// LS Electric XG5000 project: 동남140
// PLC NewPLC
// module base 0 slot 0: 입출력 모듈:XBC-DN/DP14E (DC 24V 입력 8점, 트랜지스터 출력 6점)

PROGRAM NewProgram (task: 스캔 프로그램)

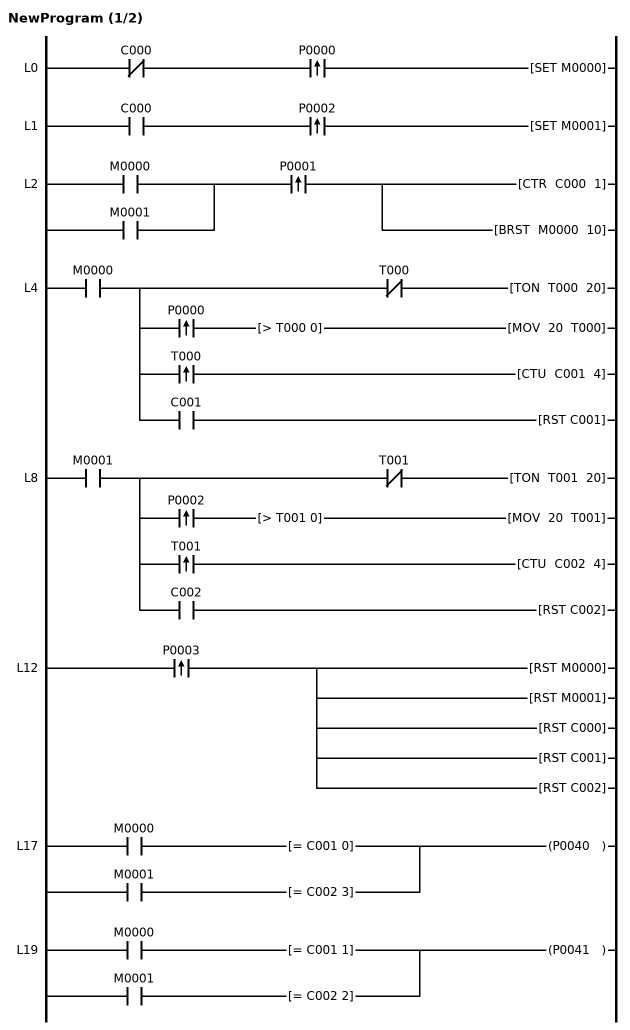
; L0
LOAD NOT  C000
ANDP      P0000
SET       M0000
; L1
LOAD      C000
ANDP      P0002
SET       M0001
; L2
LOAD      M0000
OR        M0001
ANDP      P0001
CTR       C000 1
BRST      M0000 10
; L4
LOAD      M0000
MPUSH
AND NOT   T000
TON       T000 20
MLOAD
ANDP      P0000
AND>      T000 0
MOV       20 T000
MLOAD
ANDP      T000
CTU       C001 4
MPOP
AND       C001
RST       C001
; L8
LOAD      M0001
MPUSH
AND NOT   T001
TON       T001 20
MLOAD
ANDP      P0002
AND>      T001 0
MOV       20 T001
MLOAD
ANDP      T001
CTU       C002 4
MPOP
AND       C002
RST       C002
; L12
LOADP     P0003
RST       M0000
RST       M0001
RST       C000
RST       C001
RST       C002
; L17
LOAD      M0000
AND=      C001 0
LOAD      M0001
AND=      C002 3
OR LOAD
OUT       P0040
; L19
LOAD      M0000
AND=      C001 1
LOAD      M0001
AND=      C002 2
OR LOAD
OUT       P0041

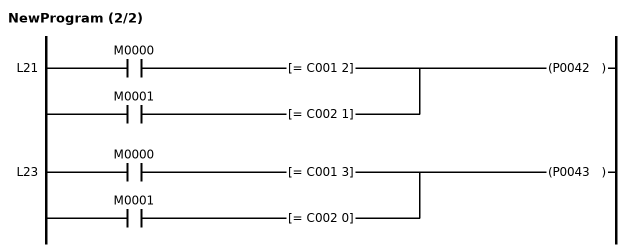
; L21
LOAD      M0000
AND=      C001 2
LOAD      M0001
AND=      C002 1
OR LOAD
OUT       P0042
; L23
LOAD      M0000
AND=      C001 3
LOAD      M0001
AND=      C002 0
OR LOAD
OUT       P0043